FUNCTION_BLOCK FB_IdBaseRecvDch EXTENDS FB_DataChannelRecvBase IMPLEMENTS I_DataChannelRecv
VAR
	/// Saber Inteface Variables
	/// -----------------------------------------------------------------
	m_pInputData: POINTER TO T_IdBase_DCH;
END_VAR

(* Copyright 2017 Cimpress

Licensed under the Apache License, Version 2.0 (the "License");
you may not use this file except in compliance with the License.
You may obtain a copy of the License at

http://www.apache.org/licenses/LICENSE-2.0

Unless required by applicable law or agreed to in writing, software
distributed under the License is distributed on an "AS IS" BASIS,
WITHOUT WARRANTIES OR CONDITIONS OF ANY KIND, either express or implied.
See the License for the specific language governing permissions and
limitations under the License. *)

SUPER^();

{attribute 'object_name' := 'InitChannel'}
METHOD InitChannel : BOOL
VAR_INPUT
	udiDataSize: UDINT;
	pInputData: POINTER TO BYTE;
END_VAR
InitChannel := FALSE;

IF udiDataSize > 0 THEN
	IF pInputData <> TC3_MEMMAN.NULL THEN
		m_uinDataSize := udiDataSize;
		m_pInputData := pInputData;
		m_eState := E_SaberPlcDHCState.Init;
		InitChannel := TRUE;
	END_IF
END_IF
END_METHOD

{attribute 'object_name' := 'GetData'}
METHOD GetData : BOOL
VAR_INPUT
	udiDataSize: UDINT;
	pData: POINTER TO BYTE;
END_VAR
GetData := FALSE;

IF m_eState = E_SaberPlcDHCState.DataReady THEN
	IF (udiDataSize > 0 ) AND (pData <> TC3_MEMMAN.NULL) THEN
		TC2_SYSTEM.MEMCPY(destAddr := pData, srcAddr := m_pInputData, n := udiDataSize);
		m_eState := E_SaberPlcDHCState.Acknowledge;	
		GetData := TRUE;
	END_IF	
END_IF
END_METHOD

END_FUNCTION_BLOCK

(* stored: Version 1.1.0.1, ProductVersion 3.1.4019.2
   POU FB_IdBaseRecvDch: Id {027a6878-45dc-4329-a3ee-28dda31b0de4}, SpecialFunc None
   Method InitChannel: Id {35fba11f-13bb-4a56-a8bf-29ffa9343d7f}
   Method GetData: Id {fde4a3d6-d56a-4699-9ab5-83ee683f7bc6} *)
